FUNCTION_BLOCK FB_CalcImageDistanceMock EXTENDS FB_FalliblePublicMock IMPLEMENTS I_CalcImageDistance
VAR
    fFocalLengthCompounded : LREAL;
END_VAR


METHOD Calculate : LREAL
VAR_INPUT
    fFocalLength	: LREAL;
    fSourceDistance	: LREAL;
END_VAR

Calculate := fFocalLengthCompounded;
END_METHOD


METHOD SetResult
VAR_INPUT
    fResult : LREAL;
END_VAR

fFocalLengthCompounded := fResult;
END_METHOD


METHOD SetValid

fFocalLengthCompounded := 1.0;
ClearError();
END_METHOD

END_FUNCTION_BLOCK

(* stored: Version 1.1.0.1
   POU FB_CalcImageDistanceMock: Id {fb46a70c-077b-4cbb-a4c8-e4e73262c8d8}, SpecialFunc None
   Method Calculate: Id {abc95be1-d404-4bee-adcd-9e1134ab5397}
   Method SetResult: Id {9f126574-7e18-4d0f-93b7-49fca5fa9b3f}
   Method SetValid: Id {ec154779-3c50-4599-8334-a67678752675} *)
